Omron CX-Programmer project NuevoProyecto (CX-Programmer 9.61)

# PLC NuevoPLC1: CQM1 CPU41

## Global symbols (name address type ; comment)
0.02 BOOL  ; S5 Tickect
0.03 BOOL  ; Reset
0.04 BOOL  ; S1
0.05 BOOL  ; S2
0.06 BOOL  ; FCin (Arriba)
0.07 BOOL  ; FCSout
0.08 BOOL  ; S3
0.09 BOOL  ; S4
0.14 BOOL  ; FCIin
0.15 BOOL  ; FCIout
100.03 BOOL  ; H2 Completo o Fuera de Servicio
100.11 BOOL  ; H1 Libre
10.00 BOOL  ; $?St$Bk?_#[2] / KA11 "Lleno"$?St$Bk?_#[2]
200.00 BOOL  ; $?St$Bk?_#[3] / "+1"$?St$Bk?_#[3]
200.01 BOOL  ; $?St$Bk?_#[4] / "-1"$?St$Bk?_#[4]
200.02 BOOL  ; $?St$Bk?_#[5] / "-1"$?St$Bk?_#[5]
20.01 BOOL  ; Estado 1
20.02 BOOL  ; Estado 2
20.03 BOOL  ; Estado 3
20.06 BOOL  ; +1
26.00 BOOL  ; Marcha
HR0 CHANNEL  ; Suma 1 coche al canal HR00
Libre 20.05 BOOL
M2_BAJAR_AUX 20.04 BOOL
PM 0.00 BOOL
PP 0.01 BOOL

## Program NuevoPrograma1 (no task)
Local symbols
CNTR001 CNT001 BOOL
EM 20.01 BOOL
Estado 20.00 BOOL  ; Estado 0
Etapa0 116.00 BOOL
Etapa1 116.01 BOOL
Etapa10 116.10 BOOL
Etapa11 116.11 BOOL
Etapa12 116.12 BOOL
Etapa13 116.13 BOOL
Etapa14 116.14 BOOL
Etapa2 116.02 BOOL
Etapa3 116.03 BOOL
Etapa4 116.04 BOOL
Etapa5 116.05 BOOL
Etapa6 116.06 BOOL
Etapa7 116.07 BOOL
Etapa8 116.08 BOOL
Etapa9 116.09 BOOL
FCIin BOOL
FCIoutSalida 0.15 BOOL
FCSin 0.06 BOOL
FCSout 0.07 BOOL
FCinSalida 0.14 BOOL
LA 100.13 BOOL  ; Lámpara de avería
LF 100.14 BOOL  ; Lámpara de funcionamiento
M11_SUBIR_AUX BOOL
M1SB 100.08 BOOL  ; Contactor marcha derecha
M1SS 100.00 BOOL  ; Contactor marcha subir
M1_BAJAR_AUX 20.02 BOOL
M1_SUBIR_AUX 20.00 BOOL
M2SB 100.15 BOOL
M2SS 100.07 BOOL
M2_SUBIR_AUX 20.03 BOOL
PMD 10.11 BOOL  ; Pulsador marcha derecha
PMI 10.10 BOOL  ; Pulsador de marcha izquierda
PP 0.01 BOOL  ; Pulsador de paro
RESET 0.03 BOOL
RT 0.13 BOOL  ; Contacto relé térmico
S_1 0.04 BOOL
S_2 0.05 BOOL
S_3 0.08 BOOL
S_4 0.09 BOOL
S_5 0.02 BOOL

### Section Sección1

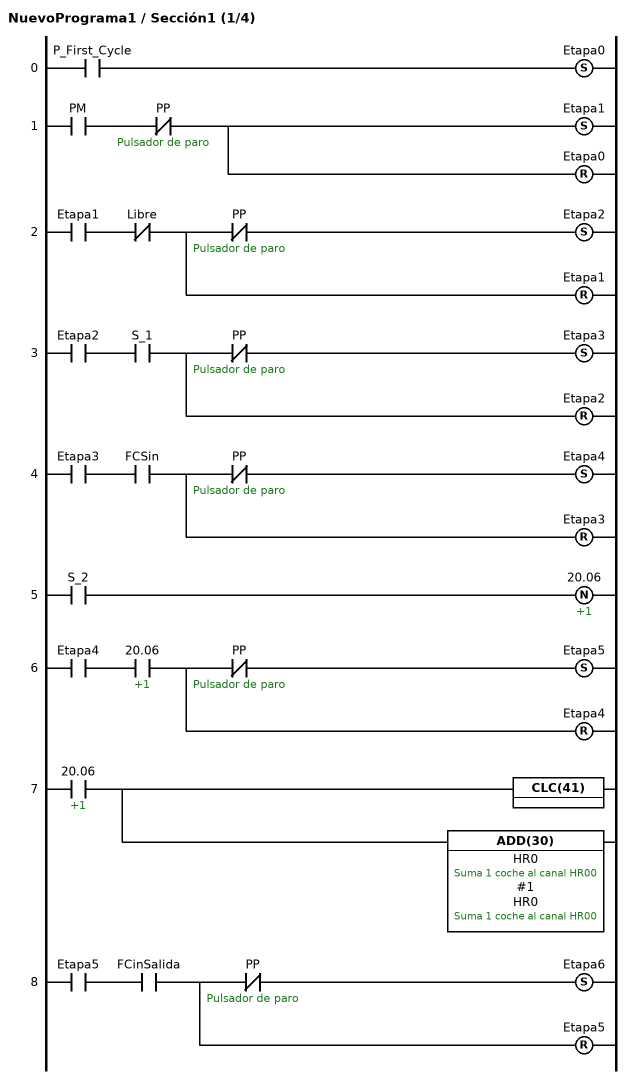
; rung 0
LD P_First_Cycle
SET Etapa0
; rung 1
LD PM
ANDNOT PP  ; Pulsador de paro
SET Etapa1
RSET Etapa0
; rung 2
LD Etapa1
ANDNOT Libre
OUT TR0
ANDNOT PP  ; Pulsador de paro
SET Etapa2
LD TR0
RSET Etapa1
; rung 3
LD Etapa2
AND S_1
OUT TR0
ANDNOT PP  ; Pulsador de paro
SET Etapa3
LD TR0
RSET Etapa2
; rung 4
LD Etapa3
AND FCSin
OUT TR0
ANDNOT PP  ; Pulsador de paro
SET Etapa4
LD TR0
RSET Etapa3
; rung 5
LD S_2
DIFD(14) 20.06  ; +1
; rung 6
LD Etapa4
AND 20.06  ; +1
OUT TR0
ANDNOT PP  ; Pulsador de paro
SET Etapa5
LD TR0
RSET Etapa4
; rung 7
LD 20.06  ; +1
CLC(41)
ADD(30) HR0 #1 HR0  ; Suma 1 coche al canal HR00
; rung 8
LD Etapa5
AND FCinSalida
OUT TR0
ANDNOT PP  ; Pulsador de paro
SET Etapa6
LD TR0
RSET Etapa5

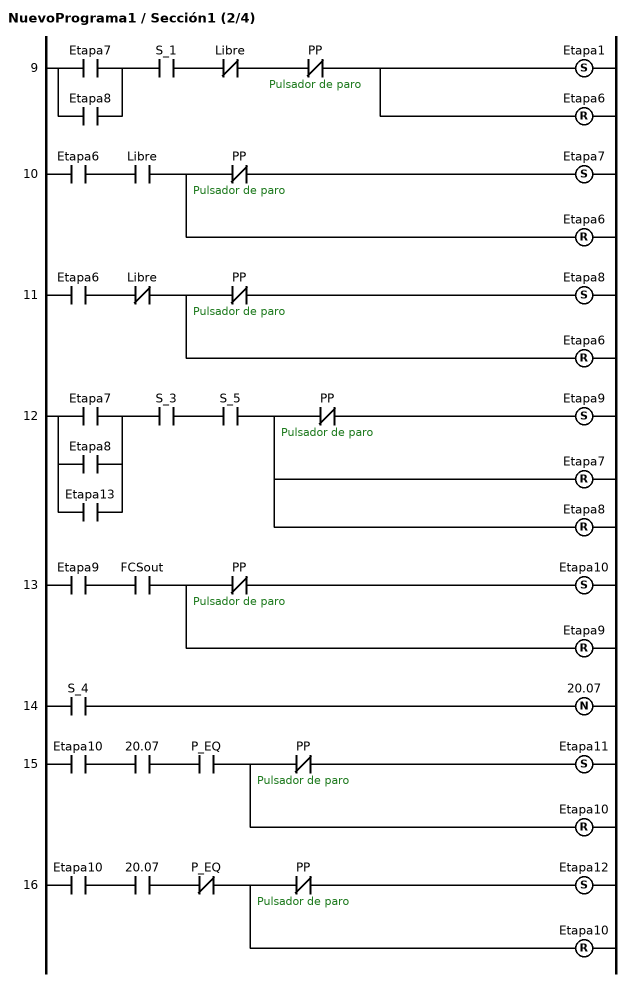
; rung 9
LD Etapa7
OR Etapa8
AND S_1
ANDNOT Libre
ANDNOT PP  ; Pulsador de paro
SET Etapa1
RSET Etapa6
; rung 10
LD Etapa6
AND Libre
OUT TR0
ANDNOT PP  ; Pulsador de paro
SET Etapa7
LD TR0
RSET Etapa6
; rung 11
LD Etapa6
ANDNOT Libre
OUT TR0
ANDNOT PP  ; Pulsador de paro
SET Etapa8
LD TR0
RSET Etapa6
; rung 12
LD Etapa7
OR Etapa8
OR Etapa13
AND S_3
AND S_5
OUT TR0
ANDNOT PP  ; Pulsador de paro
SET Etapa9
LD TR0
RSET Etapa7
RSET Etapa8
; rung 13
LD Etapa9
AND FCSout
OUT TR0
ANDNOT PP  ; Pulsador de paro
SET Etapa10
LD TR0
RSET Etapa9
; rung 14
LD S_4
DIFD(14) 20.07
; rung 15
LD Etapa10
AND 20.07
AND P_EQ
OUT TR0
ANDNOT PP  ; Pulsador de paro
SET Etapa11
LD TR0
RSET Etapa10
; rung 16
LD Etapa10
AND 20.07
ANDNOT P_EQ
OUT TR0
ANDNOT PP  ; Pulsador de paro
SET Etapa12
LD TR0
RSET Etapa10

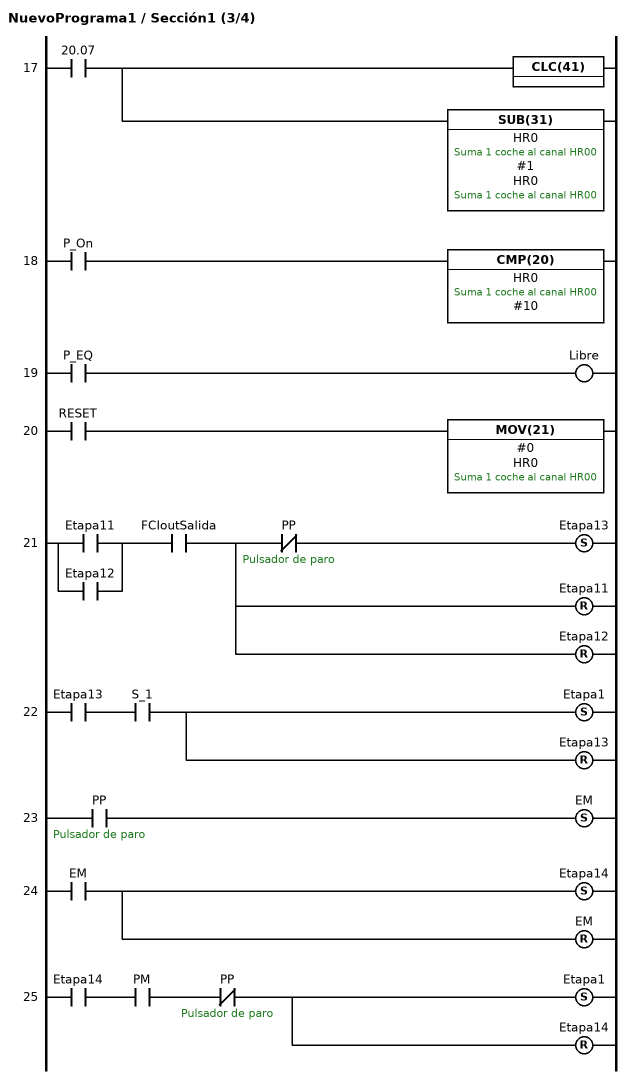
; rung 17
LD 20.07
CLC(41)
SUB(31) HR0 #1 HR0  ; Suma 1 coche al canal HR00
; rung 18
LD P_On
CMP(20) HR0 #10  ; Suma 1 coche al canal HR00
; rung 19
LD P_EQ
OUT Libre
; rung 20
LD RESET
MOV(21) #0 HR0  ; Suma 1 coche al canal HR00
; rung 21
LD Etapa11
OR Etapa12
AND FCIoutSalida
OUT TR0
ANDNOT PP  ; Pulsador de paro
SET Etapa13
LD TR0
RSET Etapa11
RSET Etapa12
; rung 22
LD Etapa13
AND S_1
SET Etapa1
RSET Etapa13
; rung 23
LD PP  ; Pulsador de paro
SET EM
; rung 24
LD EM
SET Etapa14
RSET EM
; rung 25
LD Etapa14
AND PM
ANDNOT PP  ; Pulsador de paro
SET Etapa1
RSET Etapa14

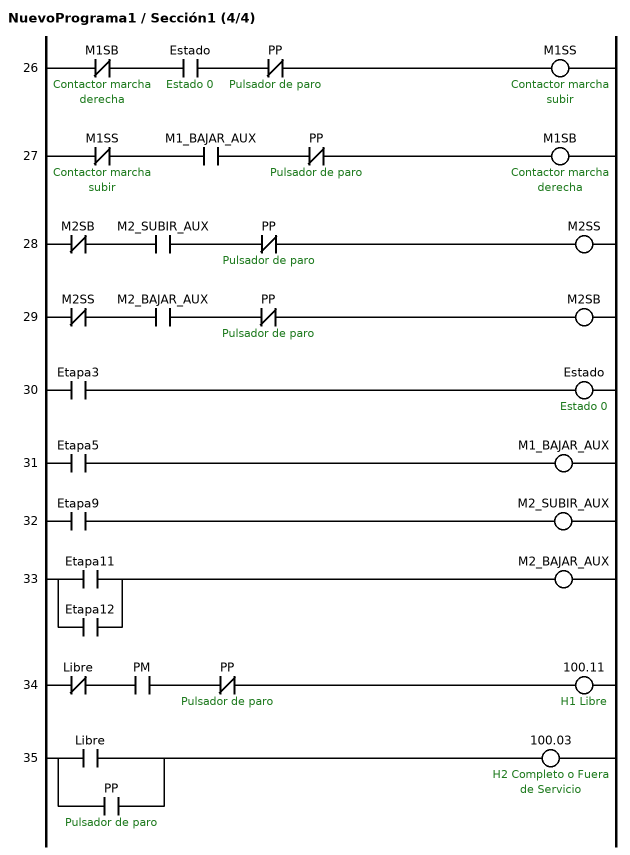
; rung 26
LDNOT M1SB  ; Contactor marcha derecha
AND Estado  ; Estado 0
ANDNOT PP  ; Pulsador de paro
OUT M1SS  ; Contactor marcha subir
; rung 27
LDNOT M1SS  ; Contactor marcha subir
AND M1_BAJAR_AUX
ANDNOT PP  ; Pulsador de paro
OUT M1SB  ; Contactor marcha derecha
; rung 28
LDNOT M2SB
AND M2_SUBIR_AUX
ANDNOT PP  ; Pulsador de paro
OUT M2SS
; rung 29
LDNOT M2SS
AND M2_BAJAR_AUX
ANDNOT PP  ; Pulsador de paro
OUT M2SB
; rung 30
LD Etapa3
OUT Estado  ; Estado 0
; rung 31
LD Etapa5
OUT M1_BAJAR_AUX
; rung 32
LD Etapa9
OUT M2_SUBIR_AUX
; rung 33
LD Etapa11
OR Etapa12
OUT M2_BAJAR_AUX
; rung 34
LDNOT Libre
AND PM
ANDNOT PP  ; Pulsador de paro
OUT 100.11  ; H1 Libre
; rung 35
LD Libre
OR PP  ; Pulsador de paro
OUT 100.03  ; H2 Completo o Fuera de Servicio

### Section END
; rung 0
END(01)